FUNCTION_BLOCK HCylinderLS (* Composite Function Block Type *)
  (* Standard: 61499-2 *)
  (* Version 0.0, 8/12/2014, valvya, nxtControl GmbH, template *)
  PACKAGE Main;
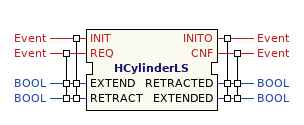
  EVENT_INPUT
    INIT WITH EXTEND, RETRACT; (* Initialization Request *)
    REQ WITH EXTEND, RETRACT; (* Normal Execution Request *)
  END_EVENT
  EVENT_OUTPUT
    INITO WITH RETRACTED, EXTENDED; (* Initialization Confirm *)
    CNF WITH RETRACTED, EXTENDED; (* Execution Confirmation *)
  END_EVENT
  VAR_INPUT
    EXTEND : BOOL; (* Input event qualifier *)
    RETRACT : BOOL;
  END_VAR
  VAR_OUTPUT
    RETRACTED : BOOL; (* Output event qualifier *)
    EXTENDED : BOOL;
  END_VAR
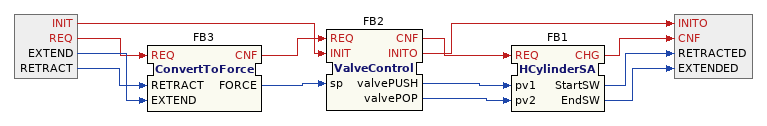
  FBS
    FB1 : HCylinderSA;
    FB2 : ValveControl;
    FB3 : ConvertToForce;
  END_FBS
  EVENT_CONNECTIONS
    FB1.CHG TO CNF;
    FB2.CNF TO FB1.REQ;
    FB2.INITO TO INITO;
    FB3.CNF TO FB2.REQ;
    REQ TO FB3.REQ;
    INIT TO FB2.INIT;
  END_CONNECTIONS
  DATA_CONNECTIONS
    FB2.valvePUSH TO FB1.pv1;
    FB2.valvePOP TO FB1.pv2;
    FB1.StartSW TO RETRACTED;
    FB1.EndSW TO EXTENDED;
    FB3.FORCE TO FB2.sp;
    RETRACT TO FB3.RETRACT;
    EXTEND TO FB3.EXTEND;
  END_CONNECTIONS
END_FUNCTION_BLOCK
